(* CoDeSys 2.3.9.41 project: lab5.pro *)
(* Libraries: STANDARD.LIB 5.6.98 11:03:02 *)

(* Task configuration *)
TASK SlowTask (PRIORITY := 2, INTERVAL := T#10ms);
	SLOW
END_TASK
TASK FastTask (PRIORITY := 1, INTERVAL := T#300ms);
	FAST
END_TASK
TASK Standard (PRIORITY := 0, INTERVAL := T#1ms);
	MAIN
END_TASK

(* POU SLOW, ST *)
PROGRAM SLOW
VAR
END_VAR
;
END_PROGRAM

(* POU FAST, ST *)
PROGRAM FAST
VAR
END_VAR
;
END_PROGRAM

(* POU MAIN, ST *)
PROGRAM MAIN
VAR
END_VAR
;
END_PROGRAM
